(* CODESYS project Parameters.library
   Company: _
   DefaultNamespace: Parameters
   Title: Parameters
   Placeholder: _Parameters
   Author: Krystian Lis et al.
   Description: No more VAR PERSITANT
   Version: 1.0.0

Project tree, tasks and I/O mapping:
  libraries: Strings, * (_)
  Persistant/
    function block BOOL_Param [ST]
    function block DINT_Param [ST]
    function block LREAL_Param [ST]
    function block REAL_Param [ST]
    function block STR_Param [ST]
    function block TIME_Param [ST]
    function block UDINT_Param [ST]
*)

// Persistant/BOOL_Param
FUNCTION_BLOCK BOOL_Param
VAR_INPUT PERSISTENT
	val				: BOOL;
END_VAR

END_FUNCTION_BLOCK

// Persistant/DINT_Param
FUNCTION_BLOCK DINT_Param
VAR_INPUT PERSISTENT
	val			: DINT;
END_VAR

END_FUNCTION_BLOCK

// Persistant/LREAL_Param
FUNCTION_BLOCK LREAL_Param
VAR_INPUT PERSISTENT
	val			: LREAL;
END_VAR

END_FUNCTION_BLOCK

// Persistant/REAL_Param
FUNCTION_BLOCK REAL_Param
VAR_INPUT PERSISTENT
	val			: REAL;
END_VAR

END_FUNCTION_BLOCK

// Persistant/STR_Param
FUNCTION_BLOCK STR_Param
VAR_INPUT PERSISTENT
	val			: Strings.Str;
END_VAR

END_FUNCTION_BLOCK

// Persistant/TIME_Param
FUNCTION_BLOCK TIME_Param
VAR_INPUT PERSISTENT
	val			: TIME;
END_VAR

END_FUNCTION_BLOCK

// Persistant/UDINT_Param
FUNCTION_BLOCK UDINT_Param
VAR_INPUT PERSISTENT
	val			: UDINT;
END_VAR

END_FUNCTION_BLOCK
